FUNCTION_BLOCK CmdValvePumpBasic (* Basic Function Block Type *)
  (* Standard: 61499-2 *)
  (* Version 0.0, 7/31/2024, Administrator, Schneider Electric, Template *)
  PACKAGE SE.Nereda;
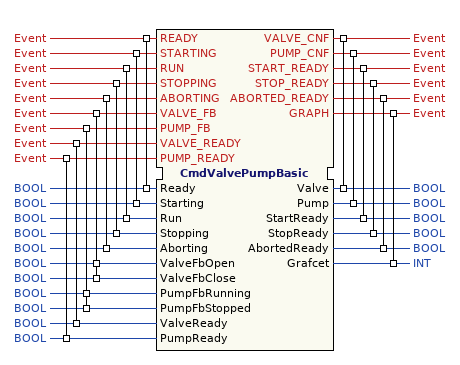
  EVENT_INPUT
    READY WITH Ready;
    STARTING WITH Starting; (* Normal Execution Request *)
    RUN WITH Run;
    STOPPING WITH Stopping;
    ABORTING WITH Aborting;
    VALVE_FB WITH ValveFbOpen, ValveFbClose;
    PUMP_FB WITH PumpFbRunning, PumpFbStopped;
    VALVE_READY WITH ValveReady;
    PUMP_READY WITH PumpReady;
  END_EVENT
  EVENT_OUTPUT
    VALVE_CNF WITH Valve; (* Execution Confirmation *)
    PUMP_CNF WITH Pump;
    START_READY WITH StartReady;
    STOP_READY WITH StopReady;
    ABORTED_READY WITH AbortedReady;
    GRAPH WITH Grafcet;
  END_EVENT
  VAR_INPUT
    Ready : BOOL;
    Starting : BOOL; (* Input event qualifier *)
    Run : BOOL;
    Stopping : BOOL;
    Aborting : BOOL;
    ValveFbOpen : BOOL;
    ValveFbClose : BOOL;
    PumpFbRunning : BOOL;
    PumpFbStopped : BOOL;
    ValveReady : BOOL;
    PumpReady : BOOL;
  END_VAR
  VAR_OUTPUT
    Valve : BOOL; (* Output event qualifier *)
    Pump : BOOL;
    StartReady : BOOL;
    StopReady : BOOL;
    AbortedReady : BOOL;
    Grafcet : INT;
  END_VAR
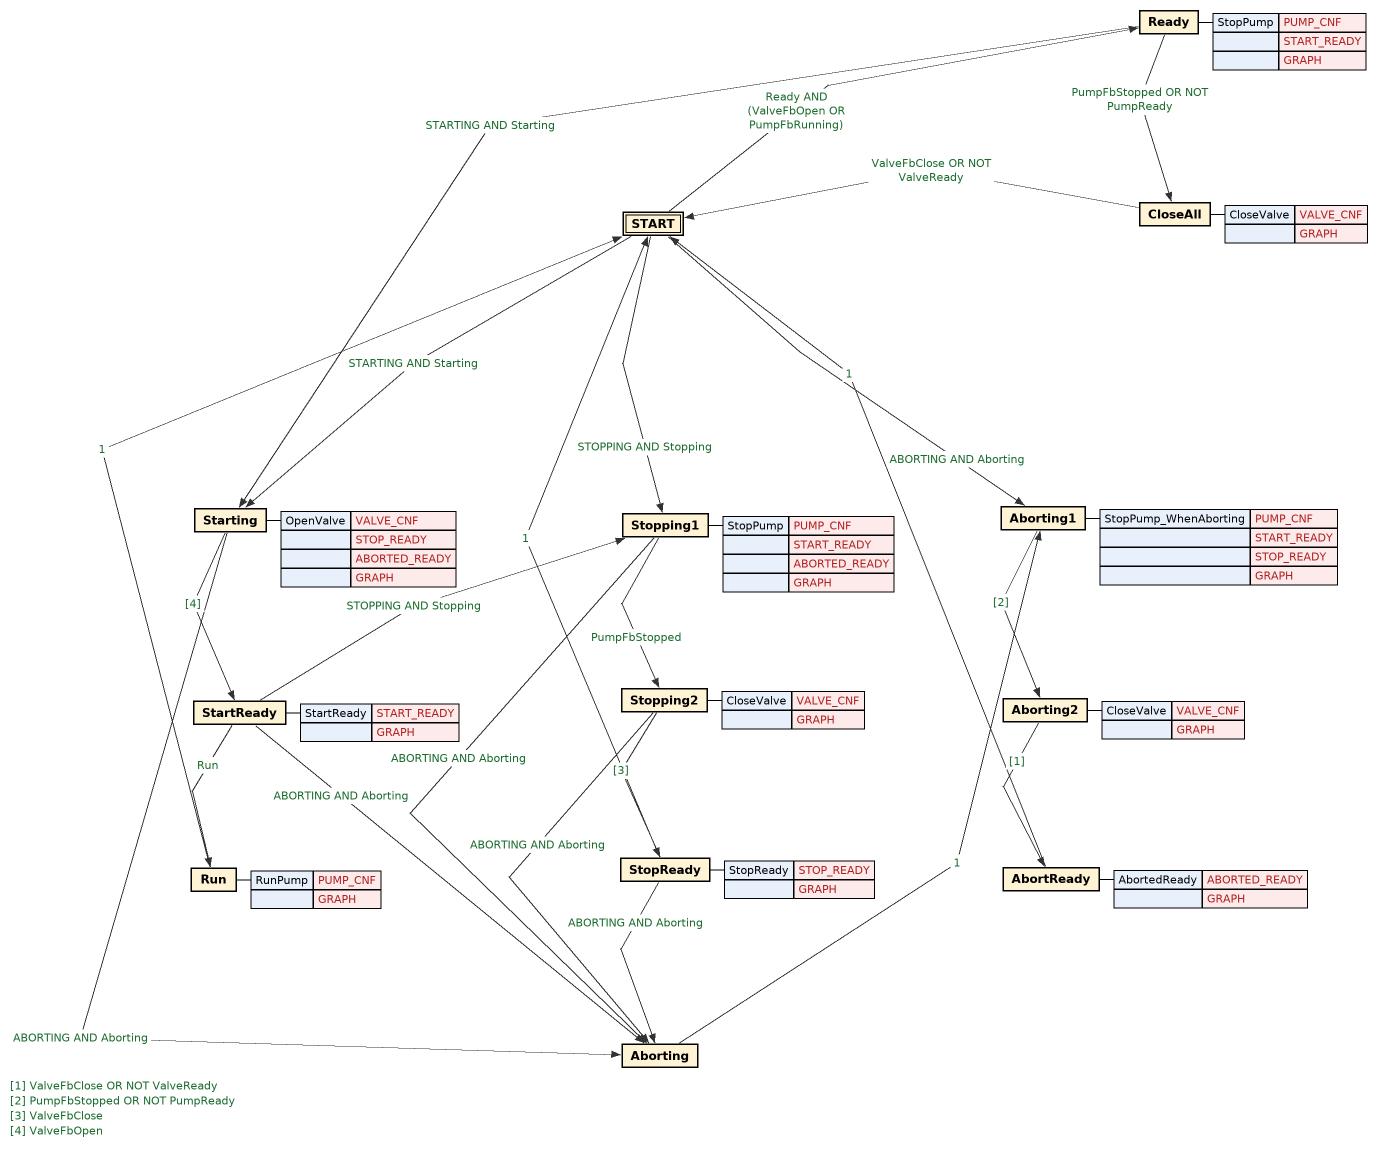
  EC_STATES
    START; (* Initial State *)
    Starting : OpenValve -> VALVE_CNF, -> STOP_READY, -> ABORTED_READY, -> GRAPH; (* Normal execution *)
    StartReady : StartReady -> START_READY, -> GRAPH;
    Stopping2 : CloseValve -> VALVE_CNF, -> GRAPH;
    StopReady : StopReady -> STOP_READY, -> GRAPH;
    Aborting2 : CloseValve -> VALVE_CNF, -> GRAPH;
    AbortReady : AbortedReady -> ABORTED_READY, -> GRAPH;
    Aborting;
    Ready : StopPump -> PUMP_CNF, -> START_READY, -> GRAPH;
    Run : RunPump -> PUMP_CNF, -> GRAPH;
    Aborting1 : StopPump_WhenAborting -> PUMP_CNF, -> START_READY, -> STOP_READY, -> GRAPH;
    Stopping1 : StopPump -> PUMP_CNF, -> START_READY, -> ABORTED_READY, -> GRAPH;
    CloseAll : CloseValve -> VALVE_CNF, -> GRAPH;
  END_STATES
  EC_TRANSITIONS
    START TO Starting := STARTING AND Starting;
    Starting TO StartReady := ValveFbOpen;
    Run TO START := 1;
    START TO Stopping1 := STOPPING AND Stopping;
    Stopping2 TO StopReady := ValveFbClose;
    StopReady TO START := 1;
    Aborting2 TO AbortReady := ValveFbClose OR NOT ValveReady;
    START TO Aborting1 := ABORTING AND Aborting;
    AbortReady TO START := 1;
    Starting TO Aborting := ABORTING AND Aborting;
    Aborting TO Aborting1 := 1;
    Stopping2 TO Aborting := ABORTING AND Aborting;
    StopReady TO Aborting := ABORTING AND Aborting;
    START TO Ready := Ready AND (ValveFbOpen OR PumpFbRunning);
    CloseAll TO START := ValveFbClose OR NOT ValveReady;
    StartReady TO Run := Run;
    StartReady TO Aborting := ABORTING AND Aborting;
    Aborting1 TO Aborting2 := PumpFbStopped OR NOT PumpReady;
    Stopping1 TO Stopping2 := PumpFbStopped;
    Ready TO CloseAll := PumpFbStopped OR NOT PumpReady;
    Stopping1 TO Aborting := ABORTING AND Aborting;
    Ready TO Starting := STARTING AND Starting;
    StartReady TO Stopping1 := STOPPING AND Stopping;
  END_TRANSITIONS
  ALGORITHM OpenValve IN ST: (* Normally executed algorithm *)
;
Grafcet := 1;
Valve := TRUE;
StopReady := FALSE;
AbortedReady := FALSE;
  END_ALGORITHM
  ALGORITHM StartReady IN ST:
;
Grafcet := 2;
StartReady := TRUE;
  END_ALGORITHM
  ALGORITHM CloseValve IN ST:
;
IF Grafcet = 4 THEN
	Grafcet := 5;
ELSIF Grafcet = 7 THEN
	Grafcet := 8;
END_IF;
Valve := FALSE;
  END_ALGORITHM
  ALGORITHM StopReady IN ST:
;
Grafcet := 6;
StopReady := TRUE;
  END_ALGORITHM
  ALGORITHM AbortedReady IN ST:
;
Grafcet := 9;
AbortedReady := TRUE;
  END_ALGORITHM
  ALGORITHM RunPump IN ST:
;
Grafcet := 3;
Pump := TRUE;
  END_ALGORITHM
  ALGORITHM StopPump IN ST:
;
Grafcet := 4;
Pump := FALSE;
StartReady := FALSE;
AbortedReady  := FALSE;
  END_ALGORITHM
  ALGORITHM StopPump_WhenAborting IN ST:
;
Grafcet := 7;
Pump := FALSE;
StartReady := FALSE;
StopReady := FALSE;
  END_ALGORITHM
END_FUNCTION_BLOCK
